{region '#Template'}
	{attribute 'Version' := '5.1.1.0'}
	{attribute 'Tags' := '"LCID": "1031", "Text": "RA, Sunprotection, Facade"'}
	{attribute 'Tags' := '"LCID": "1033", "Text": "RA, Sunprotection, Facade"'}
	{attribute 'Using' := '"Type": "Template", "URI": "Site"'}
	{attribute 'Description' := '"LCID": "1031", "Text": "Sonnenschutz Fassadendaten"'}
	{attribute 'Description' := '"LCID": "1033", "Text": "Sunprotection facade data"'}
{endregion}
// General fascade template:
// - Calculation and distribution of fascade information
FUNCTION_BLOCK FB_BA_DGWSPServer EXTENDS FB_BA_View
VAR_INPUT CONSTANT
	AdsComServerDGWS			: FB_BA_AdsComServer_DGWS;
	BuildingSunProtection		: FB_BA_BuildingSunprotection;
	arrFacade					: ARRAY[1..BA2_Param.nMaxNumberOfFacades] OF FB_BA_Facade;
END_VAR

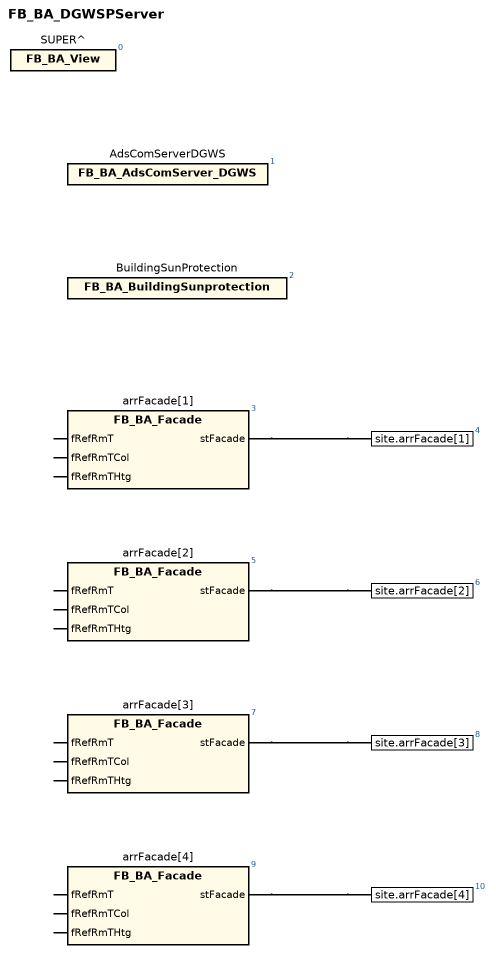
SUPER^(); // FB_BA_View
AdsComServerDGWS(); // FB_BA_AdsComServer_DGWS
BuildingSunProtection(); // FB_BA_BuildingSunprotection
arrFacade[1](); // FB_BA_Facade
site.arrFacade[1] := arrFacade[1].stFacade;
arrFacade[2](); // FB_BA_Facade
site.arrFacade[2] := arrFacade[2].stFacade;
arrFacade[3](); // FB_BA_Facade
site.arrFacade[3] := arrFacade[3].stFacade;
arrFacade[4](); // FB_BA_Facade
site.arrFacade[4] := arrFacade[4].stFacade;

METHOD FB_init : BOOL
VAR_INPUT
	bInitRetains : BOOL; // if TRUE; the retain variables are initialized (warm start / cold start)
	bInCopyCode : BOOL;  // if TRUE; the instance afterwards gets moved into the copy code (online change)
END_VAR
BuildingSunProtection.iParent				:= THIS^;	
BuildingSunProtection.iLabel				:= LblPlt_Sunlight_protection;
BuildingSunProtection.sObjectName		   	:= '{Idx=01}';
BuildingSunProtection.eDPADMode				:= E_BA_DPADMode.eInclude;

arrFacade[1].iParent			:= THIS^;	
arrFacade[1].iLabel				:= LblPlt_Facade;	
arrFacade[1].sObjectName		:= '{Idx=01}';
arrFacade[1].sDescription		:= '{Idx=01}';
arrFacade[1].eDPADMode			:= E_BA_DPADMode.eInclude;
arrFacade[1].fFcdOrtn			:= 0;	// orientation [deg] of the facade			Example: North
arrFacade[1].fFcdAngl			:= 0;	// declination [deg] of the facade
arrFacade[1].fLamWdth			:= 40;	// lamella width [mm]
arrFacade[1].fLamDstc			:= 20;	// space between two lamellas [mm]
arrFacade[1].fAzmSttRng			:= 270;	// azimuth start-range [deg] when facade is in sun
arrFacade[1].fAzmEndRng			:= 90;	// azimuth end-range [deg] when facade is in sun
arrFacade[1].fElvLoLmt			:= 0;	// elevation start-range [deg] when facade is in sun
arrFacade[1].fElvHiLmt			:= 90;	// elevation end-range [deg] when facade is in sun

arrFacade[2].iParent			:= THIS^;	
arrFacade[2].iLabel				:= LblPlt_Facade;
arrFacade[2].sObjectName		:= '{Idx=02}';
arrFacade[2].sDescription		:= '{Idx=02}';
arrFacade[2].eDPADMode			:= E_BA_DPADMode.eInclude;
arrFacade[2].fFcdOrtn			:= 90;	// orientation [deg] of the facade
arrFacade[2].fFcdAngl			:= 0;	// declination [deg] of the facade			Example: East
arrFacade[2].fLamWdth			:= 40;	// lamella width [mm]
arrFacade[2].fLamDstc			:= 20;	// space between two lamellas [mm]
arrFacade[2].fAzmSttRng			:= 0;	// azimuth start-range [deg] when facade is in sun
arrFacade[2].fAzmEndRng			:= 180;	// azimuth end-range [deg] when facade is in sun
arrFacade[2].fElvLoLmt			:= 0;	// elevation start-range [deg] when facade is in sun
arrFacade[2].fElvHiLmt			:= 90;	// elevation end-range [deg] when facade is in sun

arrFacade[3].iParent			:= THIS^;	
arrFacade[3].iLabel				:= LblPlt_Facade;
arrFacade[3].sObjectName		:= '{Idx=03}';
arrFacade[3].sDescription		:= '{Idx=03}';
arrFacade[3].eDPADMode			:= E_BA_DPADMode.eInclude;
arrFacade[3].fFcdOrtn			:= 180;	// orientation [deg] of the facade			Example: South
arrFacade[3].fFcdAngl			:= 0;	// declination [deg] of the facade
arrFacade[3].fLamWdth			:= 40;	// lamella width [mm]
arrFacade[3].fLamDstc			:= 20;	// space between two lamellas [mm]
arrFacade[3].fAzmSttRng			:= 90;	// azimuth start-range [deg] when facade is in sun
arrFacade[3].fAzmEndRng			:= 270;	// azimuth end-range [deg] when facade is in sun
arrFacade[3].fElvLoLmt			:= 0;	// elevation start-range [deg] when facade is in sun
arrFacade[3].fElvHiLmt			:= 90;	// elevation end-range [deg] when facade is in sun

arrFacade[4].iParent			:= THIS^;	
arrFacade[4].iLabel				:= LblPlt_Facade;
arrFacade[4].sObjectName		:= '{Idx=04}';
arrFacade[4].sDescription		:= '{Idx=04}';
arrFacade[4].eDPADMode			:= E_BA_DPADMode.eInclude;
arrFacade[4].fFcdOrtn			:= 270;	// orientation [deg] of the facade			Example: West
arrFacade[4].fFcdAngl			:= 0;	// declination [deg] of the facade
arrFacade[4].fLamWdth			:= 40;	// lamella width [mm]
arrFacade[4].fLamDstc			:= 20;	// space between two lamellas [mm]
arrFacade[4].fAzmSttRng			:= 180;	// azimuth start-range [deg] when facade is in sun
arrFacade[4].fAzmEndRng			:= 0;	// azimuth end-range [deg] when facade is in sun
arrFacade[4].fElvLoLmt			:= 0;	// elevation start-range [deg] when facade is in sun
arrFacade[4].fElvHiLmt			:= 90;	// elevation end-range [deg] when facade is in sun
END_METHOD

END_FUNCTION_BLOCK

(* stored: Version 1.1.0.1, ProductVersion 3.1.4024.12
   POU FB_BA_DGWSPServer: Id {c689147c-9959-4216-ae2a-7977b1138468}, SpecialFunc None
   Method FB_init: Id {48fa2802-2fa8-4529-82bd-a0c8effc5ae0} *)
